# EPICS autosave request: yaskawaBARTRobot/yaskawa_settings.req
$(P):AUTO_RUN_JOBS
